Universal Robots PolyScope program: RC_E8_PICK_820.urp

Program RC_E8_PICK_820 (createdIn=3.0.0 lastSavedIn=3.0.0 directory=/programs installation=default)
Robot Program (runOnlyOnce=true motionType=MoveJ speed=1.047198 acceleration=1.396263 useActiveTCP=false)
  'Program generated by RoboDK v4.1.0 for UR3e_HORNO on 27/07/2022 12:04:04'
  'Using nominal kinematics.'
  'Using Ref. Frame Traslado C: p[0.369000, -0.220000, 0.032000, 0.000000, 0.000000, 0.000000]'
  'Using TCP 0208-0001-0001-307-000-3 Horno: p[0.000000, 0.000000, 0.038000, 0.000000, 0.000000, 0.000000]'
  Script: set_tcp(p[0.000000, 0.000000, 0.038000, 0.000000, 0.000000, 0.000000])
  Script: movej([-0.377689, -1.963670, -0.652230, -2.094395, 1.584235, 1.239184],0.60000,0.12500,0,0.0000)
  MoveL speed 100 mm/s, acceleration 120 mm/s^2 (useActiveTCP=true)
    Waypoint Waypoint_1: TCP in base x=654 y=-474.155 z=315.972 mm, rx=0.0722 ry=3.1341 rz=0.0186 rad; joints [-21.934, -104.784, -68.076, -97.024, 90.771, 70.706] deg; flange x=653.738 y=-474.601 z=353.968 mm, rx=0.0722 ry=3.1341 rz=0.0186 rad
  'Attach to 0208-0001-0001-307-000-4 Horno'
  MoveL speed 500 mm/s, acceleration 900 mm/s^2 (useActiveTCP=true)
    Waypoint Waypoint_2: TCP in base x=658.99 y=-474.155 z=385.972 mm, rx=0.0722 ry=3.1341 rz=0.0186 rad; joints [-21.64, -112.51, -37.37, -120, 90.77, 71] deg; flange x=658.728 y=-474.601 z=423.968 mm, rx=0.0722 ry=3.1341 rz=0.0186 rad
